(* IEC 61131-3 sources: RL_MAR/experiments/comparison/autoplc/results/deepseek-ai-DeepSeek-V3.2_20260508_111905/med_88, 1 file *)

(* ---- med_88_1.st ---- *)
FUNCTION_BLOCK SmartLockerControl
VAR_INPUT
    AccessCode : INT;    (* Input for user access code *)
    LockerNumber : INT;  (* Input for selected locker number *)
END_VAR
VAR_OUTPUT
    LockerOpen : BOOL;   (* Output to control locker door *)
END_VAR
VAR
    LockerStatus : ARRAY[1..10] OF BOOL;     (* Status of individual lockers: TRUE=locked, FALSE=empty *)
    LockerAccessCode : ARRAY[1..10] OF INT;  (* Locker access codes *)
    i : INT;                                  (* Loop counter *)
    bInitialized : BOOL := FALSE;            (* Initialization flag *)
END_VAR

(* Initialize arrays only once *)
IF NOT bInitialized THEN
    (* Initialize LockerAccessCode array *)
    LockerAccessCode[1] := 1234;
    LockerAccessCode[2] := 5678;
    LockerAccessCode[3] := 9876;
    LockerAccessCode[4] := 4321;
    LockerAccessCode[5] := 6543;
    LockerAccessCode[6] := 7890;
    LockerAccessCode[7] := 3456;
    LockerAccessCode[8] := 8765;
    LockerAccessCode[9] := 2345;
    LockerAccessCode[10] := 6789;

    (* Initialize LockerStatus array - all TRUE (locked) *)
    FOR i := 1 TO 10 DO
        LockerStatus[i] := TRUE;
    END_FOR;

    bInitialized := TRUE;
END_IF;

(* Reset LockerOpen output at the beginning of each cycle *)
LockerOpen := FALSE;

(* Validate LockerNumber input *)
IF (LockerNumber >= 1) AND (LockerNumber <= 10) THEN
    (* Check if access code matches *)
    IF AccessCode = LockerAccessCode[LockerNumber] THEN
        (* Grant access and update status *)
        LockerOpen := TRUE;
        LockerStatus[LockerNumber] := FALSE;  (* Set to empty/unlocked *)
    END_IF;
END_IF;

END_FUNCTION_BLOCK
